// TIA Portal V18 export
TYPE "RecipeAxis"
   STRUCT
      Pos : Array[0..20] of Real;
      Speed : Array[0..20] of Real;
   END_STRUCT;
END_TYPE
